// Library/POUs/Calculation/MC_CalculateInverseKinematic/Structures/CalculateInverseKinematicRecvData
{attribute 'pack_mode' := '1'} 
// ------------------------------------------------------------------------- 
//  SRCI Robot Library                                                
// ------------------------------------------------------------------------- 
//                                                                           
//  Object:      CalculateInverseKinematicRecvData                                       
//  Author:      Thorsten Brach                                                
//  Date:        2024-06-09
//
//  Description:                                              
//   
//                                                                           
//  Copyright: 
//    (C) 2024 Thorsten Brach. All rights reserved                                                                                                                                            
//             Licensed under the LGPL-3.0 license.
//                                                                           
//  Disclaimer:                                                                           
//    This project is provided without any guarantee and can be used for   
//    private and commercial purposes. Any use is at the user’s 
//    own risk and responsibility.
//
// -------------------------------------------------------------------------
TYPE CalculateInverseKinematicRecvData EXTENDS RspHeader :
STRUCT
  /// Calculated robot joint position
  JointPosition      : RobotJointPosition;  
END_STRUCT
END_TYPE

// Library/POUs/Calculation/MC_CalculateInverseKinematic/Structures/CalculateInverseKinematicSendData
{attribute 'pack_mode' := '1'}
// ------------------------------------------------------------------------- 
//  SRCI Robot Library                                                
// ------------------------------------------------------------------------- 
//                                                                           
//  Object:      CalculateInverseKinematicSendData                                       
//  Author:      Thorsten Brach                                                
//  Date:        2024-06-09
//
//  Description:                                              
//   
//                                                                           
//  Copyright: 
//    (C) 2024 Thorsten Brach. All rights reserved                                                                                                                                            
//             Licensed under the LGPL-3.0 license.
//                                                                           
//  Disclaimer:                                                                           
//    This project is provided without any guarantee and can be used for   
//    private and commercial purposes. Any use is at the user’s 
//    own risk and responsibility.
//
// -------------------------------------------------------------------------
TYPE CalculateInverseKinematicSendData EXTENDS CmdHeader:   
STRUCT
  /// cartesian position
  CartesianPosition  : RobotCartesianPosition;
  /// Index of target tool
  /// • 0: Flange (default)
  /// • 1..254: Tool frames
  ToolNo             : USINT;
  /// Index of target frame
  /// • 0: WCS (default)
  /// • 1..254: User frames
  FrameNo            : USINT;  
END_STRUCT
END_TYPE

// Library/POUs/Calculation/MC_CalculateTool/Structures/CalculateToolOutCmd
{attribute 'pack_mode' := '1'} 
// ------------------------------------------------------------------------- 
//  SRCI Robot Library                                                
// ------------------------------------------------------------------------- 
//                                                                           
//  Object:      CalculateToolOutCmd                                       
//  Author:      Thorsten Brach                                                
//  Date:        2024-06-09
//
//  Description:                                              
//   
//                                                                           
//  Copyright: 
//    (C) 2024 Thorsten Brach. All rights reserved                                                                                                                                                                                                               
//             Licensed under the LGPL-3.0 license.
//                                                                           
//  Disclaimer:                                                                           
//    This project is provided without any guarantee and can be used for   
//    private and commercial purposes. Any use is at the user’s 
//    own risk and responsibility.
//
// -------------------------------------------------------------------------
TYPE CalculateToolOutCmd :
STRUCT
  /// Tool data
  ToolData           : ToolData;
  /// Maximum error of deviation of the TCP position
  /// from the fix point in world coordinate system
  /// If not supported: • -1
  TCPMaxError       : REAL;
  /// Average error of TCP position from the fix point  in world coordinate system
  /// If not supported: • -1 
  TCPMeanError      : REAL;
END_STRUCT
END_TYPE

// Library/POUs/Calculation/MC_CalculateTool/Structures/CalculateToolParCmd
{attribute 'pack_mode' := '1'} 
// ------------------------------------------------------------------------- 
//  SRCI Robot Library                                                
// ------------------------------------------------------------------------- 
//                                                                           
//  Object:      CalculateToolParCmd                                       
//  Author:      Thorsten Brach                                                
//  Date:        2024-06-09
//
//  Description:                                              
//   
//                                                                           
//  Copyright: 
//    (C) 2024 Thorsten Brach. All rights reserved                                                                                                                                      
//             Licensed under the LGPL-3.0 license.
//                                                                           
//  Disclaimer:                                                                           
//    This project is provided without any guarantee and can be used for   
//    private and commercial purposes. Any use is at the user’s 
//    own risk and responsibility.
//
// -------------------------------------------------------------------------
TYPE CalculateToolParCmd :
STRUCT
  /// Define which method should be used to calculate the tool frame
  Mode               : ToolCalculationMode;
  /// Index of target tool
  /// • 0: Flange (default)
  /// • 1..254: Tool frames
  ToolNo             : USINT;
  /// Index of target frame
  /// • 0: WCS (default)
  /// • 1..254: User frames
  FrameNo            : USINT;  
  /// • True: Tool fixed
  /// • False: Tool on flange (default)
  ExternalTCP        : BOOL;
  /// Positions in cartesian coordinates for the tool frame calculation.
  PositionsArray     : ARRAY[0..5] OF RobotCartesianPosition;
END_STRUCT
END_TYPE

// Library/POUs/Calculation/MC_CalculateTool/Structures/CalculateToolRecvData
{attribute 'pack_mode' := '1'} 
// ------------------------------------------------------------------------- 
//  SRCI Robot Library                                                
// ------------------------------------------------------------------------- 
//                                                                           
//  Object:      CalculateToolRecvData                                       
//  Author:      Thorsten Brach                                                
//  Date:        2024-06-09
//
//  Description:                                              
//   
//                                                                           
//  Copyright: 
//    (C) 2024 Thorsten Brach. All rights reserved                                                                                                                                            
//             Licensed under the LGPL-3.0 license.
//                                                                           
//  Disclaimer:                                                                           
//    This project is provided without any guarantee and can be used for   
//    private and commercial purposes. Any use is at the user’s 
//    own risk and responsibility.
//
// -------------------------------------------------------------------------
TYPE CalculateToolRecvData EXTENDS RspHeader :
STRUCT
  /// Maximum error of deviation of the TCP position
  /// from the fix point in world coordinate system
  /// If not supported: • -1
  TCPMaxError       : REAL;
  /// Average error of TCP position from the fix point  in world coordinate system
  /// If not supported: • -1 
  TCPMeanError      : REAL;
  /// Tool data
  ToolData           : ToolData;
END_STRUCT
END_TYPE

// Library/POUs/Calculation/MC_CalculateTool/Structures/CalculateToolSendData
{attribute 'pack_mode' := '1'}
// ------------------------------------------------------------------------- 
//  SRCI Robot Library                                                
// ------------------------------------------------------------------------- 
//                                                                           
//  Object:      CalculateToolSendData                                       
//  Author:      Thorsten Brach                                                
//  Date:        2024-06-09
//
//  Description:                                              
//   
//                                                                           
//  Copyright: 
//    (C) 2024 Thorsten Brach. All rights reserved                                                                                                                                            
//             Licensed under the LGPL-3.0 license.
//                                                                           
//  Disclaimer:                                                                           
//    This project is provided without any guarantee and can be used for   
//    private and commercial purposes. Any use is at the user’s 
//    own risk and responsibility.
//
// -------------------------------------------------------------------------
TYPE CalculateToolSendData EXTENDS CmdHeader:   
STRUCT
  DataIndex    : USINT;
  ///
  DataComplete : BYTE;
  /// Index of target tool
  /// • 0: Flange (default)
  /// • 1..254: Tool frames
  ToolNo       : USINT;
  /// Index of target frame
  /// • 0: WCS (default)
  /// • 1..254: User frames
  FrameNo      : USINT;    
  /// Define which method should be used to calculate the tool frame
  Mode         : ToolCalculationMode;
  /// • True: Tool fixed
  /// • False: Tool on flange (default)
  ExternalTCP  : USINT;
  /// Positions in cartesian coordinates for the tool frame calculation.
  Position     : RobotCartesianPosition;
END_STRUCT
END_TYPE

// Library/POUs/Calculation/MC_LoadMeasurementAutomatic/Structures/LoadMeasurementAutomaticOutCmd
{attribute 'pack_mode' := '1'} 
// ------------------------------------------------------------------------- 
//  SRCI Robot Library                                                
// ------------------------------------------------------------------------- 
//                                                                           
//  Object:      LoadMeasurementAutomaticOutCmd                                       
//  Author:      Thorsten Brach                                                
//  Date:        2024-06-20
//
//  Description:                                              
//   
//                                                                           
//  Copyright: 
//    (C) 2024 Thorsten Brach. All rights reserved                                                                                                                                            
//             Licensed under the LGPL-3.0 license.
//                                                                           
//  Disclaimer:                                                                           
//    This project is provided without any guarantee and can be used for   
//    private and commercial purposes. Any use is at the user’s 
//    own risk and responsibility.
//
// -------------------------------------------------------------------------
TYPE LoadMeasurementAutomaticOutCmd :
STRUCT
  /// FB is returning a unique ID for the cal led measurement.
  MeasuringID       : UINT;
  /// Measured load data (see chapter 5.5.6.4)
  LoadData          : LoadData;  
  /// Load data available
  LoadDataAvailable : BOOL;
END_STRUCT
END_TYPE

// Library/POUs/Calculation/MC_LoadMeasurementAutomatic/Structures/LoadMeasurementAutomaticParCmd
{attribute 'pack_mode' := '1'} 
// ------------------------------------------------------------------------- 
//  SRCI Robot Library                                                
// ------------------------------------------------------------------------- 
//                                                                           
//  Object:      LoadMeasurementAutomaticParCmd                                       
//  Author:      Thorsten Brach                                                
//  Date:        2024-06-20
//
//  Description:                                              
//   
//                                                                           
//  Copyright: 
//    (C) 2024 Thorsten Brach. All rights reserved                                                                                                                                            
//             Licensed under the LGPL-3.0 license.
//                                                                           
//  Disclaimer:                                                                           
//    This project is provided without any guarantee and can be used for   
//    private and commercial purposes. Any use is at the user’s 
//    own risk and responsibility.
//
// -------------------------------------------------------------------------
TYPE LoadMeasurementAutomaticParCmd :
STRUCT
  /// Define which method should be used to measure the load data
  Mode               : LoadMeasurementMode;
  /// Define which mass is expected as a result of the load measurement
  Mass               : REAL;
  /// Define the area for the allowed motion of the Joint 3. 
  /// The order of the two limit values does not matter. 
  /// Only considered with "Mode" = 0, 2.
  Area_J3            : ARRAY[0..1] OF REAL;
  /// Define the area for the allowed motion of the Joint 4. 
  /// The order of the two limit values does not matter. 
  /// Only considered with "Mode" = 0, 2.
  Area_J4            : ARRAY[0..1] OF REAL;
  /// Define the area for the allowed motion of the Joint 5. 
  /// The order of the two limit values does not matter. 
  /// Only considered with "Mode" = 0, 2.
  Area_J5            : ARRAY[0..1] OF REAL;
  /// Define the area for the allowed motion of the Joint 6. 
  /// The order of the two limit values does not matter. 
  /// Only considered with "Mode" = 0, 2.
  Area_J6            : ARRAY[0..1] OF REAL;
  /// Define the first position for the load measurement.
  /// Only considered with "Mode" = 0, 1.
  Position_1         : RobotJointPosition;
  /// Define the second position for the load measurement.
  /// Only considered with "Mode" = 3.
  Position_2         : RobotJointPosition;
  /// Define the configuration angle for the load measurement.
  /// Only considered with "Mode" = 1.
  ConfigurationAngle : REAL;
END_STRUCT
END_TYPE

// Library/POUs/Calculation/MC_LoadMeasurementAutomatic/Structures/LoadMeasurementAutomaticRecvData
{attribute 'pack_mode' := '1'} 
// ------------------------------------------------------------------------- 
//  SRCI Robot Library                                                
// ------------------------------------------------------------------------- 
//                                                                           
//  Object:      LoadMeasurementAutomaticRecvData                                       
//  Author:      Thorsten Brach                                                
//  Date:        2024-06-20
//
//  Description:                                              
//   
//                                                                           
//  Copyright: 
//    (C) 2024 Thorsten Brach. All rights reserved                                                                                                                                            
//             Licensed under the LGPL-3.0 license.
//                                                                           
//  Disclaimer:                                                                           
//    This project is provided without any guarantee and can be used for   
//    private and commercial purposes. Any use is at the user’s 
//    own risk and responsibility.
//
// -------------------------------------------------------------------------
TYPE LoadMeasurementAutomaticRecvData EXTENDS RspHeader :
STRUCT
    /// FB is returning a unique ID for the cal led measurement.
  MeasuringID       : UINT;
  /// Measured load data (see chapter 5.5.6.4)
  LoadData          : LoadData;  
  /// Load data available
  LoadDataAvailable : BOOL;
END_STRUCT
END_TYPE

// Library/POUs/Calculation/MC_LoadMeasurementAutomatic/Structures/LoadMeasurementAutomaticSendData
{attribute 'pack_mode' := '1'}
// ------------------------------------------------------------------------- 
//  SRCI Robot Library                                                
// ------------------------------------------------------------------------- 
//                                                                           
//  Object:      LoadMeasurementAutomaticSendData                                       
//  Author:      Thorsten Brach                                                
//  Date:        2024-06-20
//
//  Description:                                              
//   
//                                                                           
//  Copyright: 
//    (C) 2024 Thorsten Brach. All rights reserved                                                                                                                                            
//             Licensed under the LGPL-3.0 license.
//                                                                           
//  Disclaimer:                                                                           
//    This project is provided without any guarantee and can be used for   
//    private and commercial purposes. Any use is at the user’s 
//    own risk and responsibility.
//
// -------------------------------------------------------------------------
TYPE LoadMeasurementAutomaticSendData EXTENDS CmdHeader:   
STRUCT
    /// Define which mass is expected as a result of the load measurement
  Mass               : REAL;
  /// Define which method should be used to measure the load data
  Mode               : LoadMeasurementMode;
  /// Reserved
  Reserved           : BYTE;
  /// Define the area for the allowed motion of the Joint 3. 
  /// The order of the two limit values does not matter. 
  /// Only considered with "Mode" = 0, 2.
  Area_J3            : ARRAY[0..1] OF REAL;
  /// Define the area for the allowed motion of the Joint 4. 
  /// The order of the two limit values does not matter. 
  /// Only considered with "Mode" = 0, 2.
  Area_J4            : ARRAY[0..1] OF REAL;
  /// Define the area for the allowed motion of the Joint 5. 
  /// The order of the two limit values does not matter. 
  /// Only considered with "Mode" = 0, 2.
  Area_J5            : ARRAY[0..1] OF REAL;
  /// Define the area for the allowed motion of the Joint 6. 
  /// The order of the two limit values does not matter. 
  /// Only considered with "Mode" = 0, 2.
  Area_J6            : ARRAY[0..1] OF REAL;
  /// Define the configuration angle for the load measurement.
  /// Only considered with "Mode" = 1.
  ConfigurationAngle : REAL;
  /// Define the first position for the load measurement.
  /// Only considered with "Mode" = 0, 1.
  Position_1         : RobotJointPosition;
  /// Define the second position for the load measurement.
  /// Only considered with "Mode" = 3.
  Position_2         : RobotJointPosition;
END_STRUCT
END_TYPE

// Library/POUs/Calculation/MC_LoadMeasurementSequential/Structures/LoadMeasurementSequentialOutCmd
{attribute 'pack_mode' := '1'} 
// ------------------------------------------------------------------------- 
//  SRCI Robot Library                                                
// ------------------------------------------------------------------------- 
//                                                                           
//  Object:      LoadMeasurementSequentialOutCmd                                       
//  Author:      Thorsten Brach                                                
//  Date:        2024-06-20
//
//  Description:                                              
//   
//                                                                           
//  Copyright: 
//    (C) 2024 Thorsten Brach. All rights reserved                                                                                                                                            
//             Licensed under the LGPL-3.0 license.
//                                                                           
//  Disclaimer:                                                                           
//    This project is provided without any guarantee and can be used for   
//    private and commercial purposes. Any use is at the user’s 
//    own risk and responsibility.
//
// -------------------------------------------------------------------------
TYPE LoadMeasurementSequentialOutCmd :
STRUCT
  /// FB is returning a unique ID for the cal led measurement.
  MeasuringID        : UINT;
  /// Measured load data (see chapter 5.5.6.4)
  LoadData           : LoadData;
  /// Load data available
  LoadDataAvailable : BOOL;
END_STRUCT
END_TYPE

// Library/POUs/Calculation/MC_LoadMeasurementSequential/Structures/LoadMeasurementSequentialParCmd
{attribute 'pack_mode' := '1'} 
// ------------------------------------------------------------------------- 
//  SRCI Robot Library                                                
// ------------------------------------------------------------------------- 
//                                                                           
//  Object:      LoadMeasurementSequentialParCmd                                       
//  Author:      Thorsten Brach                                                
//  Date:        2024-06-20
//
//  Description:                                              
//   
//                                                                           
//  Copyright: 
//    (C) 2024 Thorsten Brach. All rights reserved                                                                                                                                            
//             Licensed under the LGPL-3.0 license.
//                                                                           
//  Disclaimer:                                                                           
//    This project is provided without any guarantee and can be used for   
//    private and commercial purposes. Any use is at the user’s 
//    own risk and responsibility.
//
// -------------------------------------------------------------------------
TYPE LoadMeasurementSequentialParCmd :
STRUCT
  /// Define which step of the load estimation should be executed:
  Mode               : LoadMeasurementSteps;
  /// Define which mass is expected as a result of the load measurement
  Mass               : REAL;
END_STRUCT
END_TYPE

// Library/POUs/Calculation/MC_LoadMeasurementSequential/Structures/LoadMeasurementSequentialRecvData
{attribute 'pack_mode' := '1'} 
// ------------------------------------------------------------------------- 
//  SRCI Robot Library                                                
// ------------------------------------------------------------------------- 
//                                                                           
//  Object:      LoadMeasurementSequentialRecvData                                       
//  Author:      Thorsten Brach                                                
//  Date:        2024-06-20
//
//  Description:                                              
//   
//                                                                           
//  Copyright: 
//    (C) 2024 Thorsten Brach. All rights reserved                                                                                                                                            
//             Licensed under the LGPL-3.0 license.
//                                                                           
//  Disclaimer:                                                                           
//    This project is provided without any guarantee and can be used for   
//    private and commercial purposes. Any use is at the user’s 
//    own risk and responsibility.
//
// -------------------------------------------------------------------------
TYPE LoadMeasurementSequentialRecvData EXTENDS RspHeader :
STRUCT
  /// FB is returning a unique ID for the cal led measurement.
  MeasuringID       : UINT;
  /// Measured load data (see chapter 5.5.6.4)
  LoadData          : LoadData;  
  /// Load data available
  LoadDataAvailable : BOOL;
END_STRUCT
END_TYPE

// Library/POUs/Calculation/MC_LoadMeasurementSequential/Structures/LoadMeasurementSequentialSendData
{attribute 'pack_mode' := '1'}
// ------------------------------------------------------------------------- 
//  SRCI Robot Library                                                
// ------------------------------------------------------------------------- 
//                                                                           
//  Object:      LoadMeasurementSequentialSendData                                       
//  Author:      Thorsten Brach                                                
//  Date:        2024-06-20
//
//  Description:                                              
//   
//                                                                           
//  Copyright: 
//    (C) 2024 Thorsten Brach. All rights reserved                                                                                                                                            
//             Licensed under the LGPL-3.0 license.
//                                                                           
//  Disclaimer:                                                                           
//    This project is provided without any guarantee and can be used for   
//    private and commercial purposes. Any use is at the user’s 
//    own risk and responsibility.
//
// -------------------------------------------------------------------------
TYPE LoadMeasurementSequentialSendData EXTENDS CmdHeader:   
STRUCT
    /// Define which mass is expected as a result of the load measurement
  Mass               : REAL;
  /// Define which step of the load estimation should be executed:
  Mode               : LoadMeasurementSteps;
END_STRUCT
END_TYPE

// Library/POUs/ConveyorTracking/MC_ActivateConveyorTracking/Structures/ActivateConveyorTrackingOutCmd
{attribute 'pack_mode' := '1'} 
// ------------------------------------------------------------------------- 
//  SRCI Robot Library                                                
// ------------------------------------------------------------------------- 
//                                                                           
//  Object:      ActivateConveyorTrackingOutCmd                                       
//  Author:      Thorsten Brach                                                
//  Date:        2024-06-11
//
//  Description:                                              
//   
//                                                                           
//  Copyright: 
//    (C) 2024 Thorsten Brach. All rights reserved                                                                                                                                                                                                               
//             Licensed under the LGPL-3.0 license.
//                                                                           
//  Disclaimer:                                                                           
//    This project is provided without any guarantee and can be used for   
//    private and commercial purposes. Any use is at the user’s 
//    own risk and responsibility.
//
// -------------------------------------------------------------------------
TYPE ActivateConveyorTrackingOutCmd :
STRUCT
  /// Current status of "ConveyorTracking" according to Table 6-432
  TrackingStatus     : TrackingStatus;
  /// Relates to "ConnectionMode" 1 – "RC connected": Traveled distance of assigned conveyor since ConveyorTracking has been activated (offset)
  RCEncoderValue     : REAL;
END_STRUCT
END_TYPE

// Library/POUs/ConveyorTracking/MC_ActivateConveyorTracking/Structures/ActivateConveyorTrackingParCmd
{attribute 'pack_mode' := '1'} 
// ------------------------------------------------------------------------- 
//  SRCI Robot Library                                                
// ------------------------------------------------------------------------- 
//                                                                           
//  Object:      ActivateConveyorTrackingParCmd                                       
//  Author:      Thorsten Brach                                                
//  Date:        2024-06-11
//
//  Description:                                              
//   
//                                                                           
//  Copyright: 
//    (C) 2024 Thorsten Brach. All rights reserved                                                                                                                                      
//             Licensed under the LGPL-3.0 license.
//                                                                           
//  Disclaimer:                                                                           
//    This project is provided without any guarantee and can be used for   
//    private and commercial purposes. Any use is at the user’s 
//    own risk and responsibility.
//
// -------------------------------------------------------------------------
TYPE ActivateConveyorTrackingParCmd :
STRUCT
  /// Index of assigned conveyor
  ConveyorNo         : SINT;
  /// Specifies encoder connection setup (at least one option must be supported)
  ConnectionMode     : ConnectionMode;
  /// Relates to "ConnectionMode" 1 – "PLC connected": Value of the encoder connected to the conveyor belt
  PLCEncoderValue    : REAL;
END_STRUCT
END_TYPE

// Library/POUs/ConveyorTracking/MC_ActivateConveyorTracking/Structures/ActivateConveyorTrackingRecvData
{attribute 'pack_mode' := '1'} 
// ------------------------------------------------------------------------- 
//  SRCI Robot Library                                                
// ------------------------------------------------------------------------- 
//                                                                           
//  Object:      ActivateConveyorTrackingRecvData                                       
//  Author:      Thorsten Brach                                                
//  Date:        2024-06-11
//
//  Description:                                              
//   
//                                                                           
//  Copyright: 
//    (C) 2024 Thorsten Brach. All rights reserved                                                                                                                                            
//             Licensed under the LGPL-3.0 license.
//                                                                           
//  Disclaimer:                                                                           
//    This project is provided without any guarantee and can be used for   
//    private and commercial purposes. Any use is at the user’s 
//    own risk and responsibility.
//
// -------------------------------------------------------------------------
TYPE ActivateConveyorTrackingRecvData EXTENDS RspHeader :
STRUCT
  /// Maximum error of deviation of the TCP position
  /// from the fix point in world coordinate system
  /// If not supported: • -1
  TrackingStatus : TrackingStatus;
END_STRUCT
END_TYPE

// Library/POUs/ConveyorTracking/MC_ActivateConveyorTracking/Structures/ActivateConveyorTrackingSendData
{attribute 'pack_mode' := '1'}
// ------------------------------------------------------------------------- 
//  SRCI Robot Library                                                
// ------------------------------------------------------------------------- 
//                                                                           
//  Object:      ActivateConveyorTrackingSendData                                       
//  Author:      Thorsten Brach                                                
//  Date:        2024-06-11
//
//  Description:                                              
//   
//                                                                           
//  Copyright: 
//    (C) 2024 Thorsten Brach. All rights reserved                                                                                                                                            
//             Licensed under the LGPL-3.0 license.
//                                                                           
//  Disclaimer:                                                                           
//    This project is provided without any guarantee and can be used for   
//    private and commercial purposes. Any use is at the user’s 
//    own risk and responsibility.
//
// -------------------------------------------------------------------------
TYPE ActivateConveyorTrackingSendData EXTENDS CmdHeader:   
STRUCT
  /// Index of assigned conveyor
  ConveyorNo     : SINT;
  /// Specifies encoder connection setup (at least one option must be supported)
  ConnectionMode : SINT;
END_STRUCT
END_TYPE

// Library/POUs/ConveyorTracking/MC_ConfigureConveyor/Structures/ConfigureConveyorOutCmd
{attribute 'pack_mode' := '1'} 
// ------------------------------------------------------------------------- 
//  SRCI Robot Library                                                
// ------------------------------------------------------------------------- 
//                                                                           
//  Object:      ConfigureConveyorOutCmd                                       
//  Author:      Thorsten Brach                                                
//  Date:        2024-06-11
//
//  Description:                                              
//   
//                                                                           
//  Copyright: 
//    (C) 2024 Thorsten Brach. All rights reserved                                                                                                                                                                                                               
//             Licensed under the LGPL-3.0 license.
//                                                                           
//  Disclaimer:                                                                           
//    This project is provided without any guarantee and can be used for   
//    private and commercial purposes. Any use is at the user’s 
//    own risk and responsibility.
//
// -------------------------------------------------------------------------
TYPE ConfigureConveyorOutCmd :
STRUCT
END_STRUCT
END_TYPE

// Library/POUs/ConveyorTracking/MC_ConfigureConveyor/Structures/ConfigureConveyorParCmd
{attribute 'pack_mode' := '1'} 
// ------------------------------------------------------------------------- 
//  SRCI Robot Library                                                
// ------------------------------------------------------------------------- 
//                                                                           
//  Object:      ConfigureConveyorParCmd                                       
//  Author:      Thorsten Brach                                                
//  Date:        2024-06-11
//
//  Description:                                              
//   
//                                                                           
//  Copyright: 
//    (C) 2024 Thorsten Brach. All rights reserved                                                                                                                                      
//             Licensed under the LGPL-3.0 license.
//                                                                           
//  Disclaimer:                                                                           
//    This project is provided without any guarantee and can be used for   
//    private and commercial purposes. Any use is at the user’s 
//    own risk and responsibility.
//
// -------------------------------------------------------------------------
TYPE ConfigureConveyorParCmd :
STRUCT
  /// Index of assigned conveyor
  ConveyorNo         : USINT;  
  ///Define the origin coordinate system of the conveyor belt, with the X-Axis pointing in the direction of the movement of the conveyor belt.
  ConveyorOrigin     : FrameData;
  /// Define the type of the conveyor
  ConveyorType       : ConveyorType;
  /// Relates to "ConveyorType" "Circular Tracking": Define the radius of the circular conveyor
  Radius             : REAL;
  /// Distance [mm] from the origin of the conveyor belt to the beginning of the "SyncInZone"
  StartDistance      : REAL;
  /// Distance [mm] from the origin of the conveyor belt to the end of the "SyncOutZone"
  EndDistance        : REAL;
  /// Define the length of the "SyncInZone"
  SyncInLength       : REAL;
  /// Define the length of the "SyncOutZone"
  SyncOutLength      : REAL;
END_STRUCT
END_TYPE

// Library/POUs/ConveyorTracking/MC_ConfigureConveyor/Structures/ConfigureConveyorRecvData
{attribute 'pack_mode' := '1'} 
// ------------------------------------------------------------------------- 
//  SRCI Robot Library                                                
// ------------------------------------------------------------------------- 
//                                                                           
//  Object:      ConfigureConveyorRecvData                                       
//  Author:      Thorsten Brach                                                
//  Date:        2024-06-11
//
//  Description:                                              
//   
//                                                                           
//  Copyright: 
//    (C) 2024 Thorsten Brach. All rights reserved                                                                                                                                            
//             Licensed under the LGPL-3.0 license.
//                                                                           
//  Disclaimer:                                                                           
//    This project is provided without any guarantee and can be used for   
//    private and commercial purposes. Any use is at the user’s 
//    own risk and responsibility.
//
// -------------------------------------------------------------------------
TYPE ConfigureConveyorRecvData EXTENDS RspHeader :
STRUCT
END_STRUCT
END_TYPE

// Library/POUs/ConveyorTracking/MC_ConfigureConveyor/Structures/ConfigureConveyorSendData
{attribute 'pack_mode' := '1'}
// ------------------------------------------------------------------------- 
//  SRCI Robot Library                                                
// ------------------------------------------------------------------------- 
//                                                                           
//  Object:      ConfigureConveyorSendData                                       
//  Author:      Thorsten Brach                                                
//  Date:        2024-06-11
//
//  Description:                                              
//   
//                                                                           
//  Copyright: 
//    (C) 2024 Thorsten Brach. All rights reserved                                                                                                                                            
//             Licensed under the LGPL-3.0 license.
//                                                                           
//  Disclaimer:                                                                           
//    This project is provided without any guarantee and can be used for   
//    private and commercial purposes. Any use is at the user’s 
//    own risk and responsibility.
//
// -------------------------------------------------------------------------
TYPE ConfigureConveyorSendData EXTENDS CmdHeader:   
STRUCT
  ///Define the origin coordinate system of the conveyor belt, with the X-Axis pointing in the direction of the movement of the conveyor belt.
  ConveyorOrigin          : FrameData;
  /// ConveyorOrigin available
  ConveyorOriginAvailable : BOOL;
  /// Index of assigned conveyor
  ConveyorNo              : USINT;  
  /// Define the type of the conveyor
  ConveyorType            : ConveyorType;
  /// Relates to "ConveyorType" "Circular Tracking": Define the radius of the circular conveyor
  Radius                  : REAL;
  /// Distance [mm] from the origin of the conveyor belt to the beginning of the "SyncInZone"
  StartDistance           : REAL;
  /// Distance [mm] from the origin of the conveyor belt to the end of the "SyncOutZone"
  EndDistance             : REAL;
  /// Define the length of the "SyncInZone"
  SyncInLength            : REAL;
  /// Define the length of the "SyncOutZone"
  SyncOutLength           : REAL;
END_STRUCT
END_TYPE

// Library/POUs/ConveyorTracking/MC_RedefineTrackingPos/Structures/RedefineTrackingPosOutCmd
{attribute 'pack_mode' := '1'} 
// ------------------------------------------------------------------------- 
//  SRCI Robot Library                                                
// ------------------------------------------------------------------------- 
//                                                                           
//  Object:      RedefineTrackingPosOutCmd                                       
//  Author:      Thorsten Brach                                                
//  Date:        2024-06-11
//
//  Description:                                              
//   
//                                                                           
//  Copyright: 
//    (C) 2024 Thorsten Brach. All rights reserved                                                                                                                                                                                                               
//             Licensed under the LGPL-3.0 license.
//                                                                           
//  Disclaimer:                                                                           
//    This project is provided without any guarantee and can be used for   
//    private and commercial purposes. Any use is at the user’s 
//    own risk and responsibility.
//
// -------------------------------------------------------------------------
TYPE RedefineTrackingPosOutCmd :
STRUCT
  /// Unique system-generated ID of the "Action" when the function is triggered.
  /// • >0: The "Action" is started by the trigger funcrion with identical FollowID.
  /// • <0: The "Action" is stopped by the trigger function with identical FollowID.
  /// For more information see chapter 5.5.12.4 EmitterID, ListenerID, FollowID and OriginID
  OriginID               : INT;
  /// Relates to ListenerID >0
  /// Number of successful trigger-based command invocations - For more information refer TO chapter 5.5.12.4
  InvocationCounter      : USINT;  
END_STRUCT
END_TYPE

// Library/POUs/ConveyorTracking/MC_RedefineTrackingPos/Structures/RedefineTrackingPosParCmd
{attribute 'pack_mode' := '1'} 
// ------------------------------------------------------------------------- 
//  SRCI Robot Library                                                
// ------------------------------------------------------------------------- 
//                                                                           
//  Object:      RedefineTrackingPosParCmd                                       
//  Author:      Thorsten Brach                                                
//  Date:        2024-06-11
//
//  Description:                                              
//   
//                                                                           
//  Copyright: 
//    (C) 2024 Thorsten Brach. All rights reserved                                                                                                                                      
//             Licensed under the LGPL-3.0 license.
//                                                                           
//  Disclaimer:                                                                           
//    This project is provided without any guarantee and can be used for   
//    private and commercial purposes. Any use is at the user’s 
//    own risk and responsibility.
//
// -------------------------------------------------------------------------
TYPE RedefineTrackingPosParCmd :
STRUCT
  /// Relates to ListenerID >0:
  ProcessingMode         : ProcessingMode;
  /// Index of assigned conveyor
  ConveyorNo             : USINT;
  /// Relates to ListenerID = 0:
  /// Define initial work piece position relative to the conveyor belt origin:
  /// • Origin (X, Y, Z in mm)
  /// • Orientation (RX, RY, RZ in degree)
  /// For more information refer to chapter 5.5.14.
  InitObjectPosition     : ARRAY[0..5] OF REAL;
  /// Relates to ListenerID = 0:
  /// Travel distance of assigned UCS between work piece detection (InitObjectPosition) and execution of this command.
  TrackingOffset         : REAL;
  /// Relates to ListenerID >0
  /// Start index of real registers containing InitObjectPosition for trigger-based execution.
  StartIndexInitPosition : USINT;
  /// Define the index number of the UCS that is assigned to the conveyor by the function "ConveyorTracking".
  /// For more information refer to chapter 5.5.14.
  FrameNo                : USINT;
  /// Relates to ListenerID >0
  /// Index of real register containing TrackingOffset for trigger-based execution
  IndexTrackingOffset    : USINT;
  /// ID of associated trigger function:
  /// • 0: No Trigger (default): No trigger related behavior
  /// • >0: Trigger: o Start executing, when the trigger function with the identical EmitterID is triggered.
  /// Always positive.
  /// For more information, see chapter 5.5.12 Triggers
  ListenerID             :  SINT;
END_STRUCT
END_TYPE

// Library/POUs/ConveyorTracking/MC_RedefineTrackingPos/Structures/RedefineTrackingPosRecvData
{attribute 'pack_mode' := '1'} 
// ------------------------------------------------------------------------- 
//  SRCI Robot Library                                                
// ------------------------------------------------------------------------- 
//                                                                           
//  Object:      RedefineTrackingPosRecvData                                       
//  Author:      Thorsten Brach                                                
//  Date:        2024-06-11
//
//  Description:                                              
//   
//                                                                           
//  Copyright: 
//    (C) 2024 Thorsten Brach. All rights reserved                                                                                                                                            
//             Licensed under the LGPL-3.0 license.
//                                                                           
//  Disclaimer:                                                                           
//    This project is provided without any guarantee and can be used for   
//    private and commercial purposes. Any use is at the user’s 
//    own risk and responsibility.
//
// -------------------------------------------------------------------------
TYPE RedefineTrackingPosRecvData EXTENDS RspHeader :
STRUCT
  
  InvocationCounter : USINT;
  /// Reserve
  Reserved          : SINT;
  /// Unique system-generated ID of the "Action" when the function is triggered.
  /// • >0: The "Action" is started by the trigger funcrion with identical FollowID.
  /// • <0: The "Action" is stopped by the trigger function with identical FollowID.
  /// For more information see chapter 5.5.12.4 EmitterID, ListenerID, FollowID and OriginID
  OriginID          : INT;
END_STRUCT
END_TYPE

// Library/POUs/ConveyorTracking/MC_RedefineTrackingPos/Structures/RedefineTrackingPosSendData
{attribute 'pack_mode' := '1'}
// ------------------------------------------------------------------------- 
//  SRCI Robot Library                                                
// ------------------------------------------------------------------------- 
//                                                                           
//  Object:      RedefineTrackingPosSendData                                       
//  Author:      Thorsten Brach                                                
//  Date:        2024-06-11
//
//  Description:                                              
//   
//                                                                           
//  Copyright: 
//    (C) 2024 Thorsten Brach. All rights reserved                                                                                                                                            
//             Licensed under the LGPL-3.0 license.
//                                                                           
//  Disclaimer:                                                                           
//    This project is provided without any guarantee and can be used for   
//    private and commercial purposes. Any use is at the user’s 
//    own risk and responsibility.
//
// -------------------------------------------------------------------------
TYPE RedefineTrackingPosSendData EXTENDS CmdHeader:   
STRUCT
  /// EmitterID
  EmitterID              : ARRAY[0..3] OF SINT;
  /// ID of associated trigger function:
  /// • 0: No Trigger (default): No trigger related behavior
  /// • >0: Trigger: o Start executing, when the trigger function with the identical EmitterID is triggered.
  /// Always positive.
  /// For more information, see chapter 5.5.12 Triggers
  ListenerID             : SINT;
  /// Reserve
  Reserve                : BYTE;
  /// Index of assigned conveyor
  ConveyorNo             : USINT;
  /// Relates to ListenerID >0
  /// Start index of real registers containing InitObjectPosition for trigger-based execution.
  StartIndexInitPosition : USINT;
  /// Relates to ListenerID = 0:
  /// Travel distance of assigned UCS between work piece detection (InitObjectPosition) and execution of this command.
  TrackingOffset         : REAL;
  /// Define the index number of the UCS that is assigned to the conveyor by the function "ConveyorTracking".
  /// For more information refer to chapter 5.5.14.
  FrameNo                : USINT;
  /// Relates to ListenerID >0
  /// Index of real register containing TrackingOffset for trigger-based execution
  IndexTrackingOffset    : USINT;
END_STRUCT
END_TYPE

// Library/POUs/ConveyorTracking/MC_SyncToConveyor/Structures/SyncToConveyorOutCmd
{attribute 'pack_mode' := '1'} 
// ------------------------------------------------------------------------- 
//  SRCI Robot Library                                                
// ------------------------------------------------------------------------- 
//                                                                           
//  Object:      SyncToConveyorOutCmd                                       
//  Author:      Thorsten Brach                                                
//  Date:        2024-06-11
//
//  Description:                                              
//   
//                                                                           
//  Copyright: 
//    (C) 2024 Thorsten Brach. All rights reserved                                                                                                                                                                                                               
//             Licensed under the LGPL-3.0 license.
//                                                                           
//  Disclaimer:                                                                           
//    This project is provided without any guarantee and can be used for   
//    private and commercial purposes. Any use is at the user’s 
//    own risk and responsibility.
//
// -------------------------------------------------------------------------
TYPE SyncToConveyorOutCmd :
STRUCT
  /// Relates to ListenerID >0
  /// Number of successful trigger-based command invocations - For more information refer TO chapter 5.5.12.4
  InvocationCounter      : USINT;  
  /// Reserve
  Reserve                : BYTE;
  /// Unique system-generated ID of the "Action" when the function is triggered.
  /// • >0: The "Action" is started by the trigger funcrion with identical FollowID.
  /// • <0: The "Action" is stopped by the trigger function with identical FollowID.
  /// For more information see chapter 5.5.12.4 EmitterID, ListenerID, FollowID and OriginID
  OriginID               : INT;
  /// The TCP is in synchronization with the object on the conveyor belt.
  InSync                 : BOOL;
END_STRUCT
END_TYPE

// Library/POUs/ConveyorTracking/MC_SyncToConveyor/Structures/SyncToConveyorParCmd
{attribute 'pack_mode' := '1'} 
// ------------------------------------------------------------------------- 
//  SRCI Robot Library                                                
// ------------------------------------------------------------------------- 
//                                                                           
//  Object:      SyncToConveyorParCmd                                       
//  Author:      Thorsten Brach                                                
//  Date:        2024-06-11
//
//  Description:                                              
//   
//                                                                           
//  Copyright: 
//    (C) 2024 Thorsten Brach. All rights reserved                                                                                                                                      
//             Licensed under the LGPL-3.0 license.
//                                                                           
//  Disclaimer:                                                                           
//    This project is provided without any guarantee and can be used for   
//    private and commercial purposes. Any use is at the user’s 
//    own risk and responsibility.
//
// -------------------------------------------------------------------------
TYPE SyncToConveyorParCmd :
STRUCT
  /// Index of assigned conveyor
  ConveyorNo      : USINT;
  /// Define the index number of the UCS that will be assigned to the conveyor.
  /// For more information refer to chapter 5.5.14
  FrameNo         : USINT;
  /// Defines when synchronization starts.
  SyncInMode      : SyncInMode;
  /// Relates to "SyncInMode" "After distance" (1) and "After time" (2):
  /// Parameter for the synchronization
  /// • "After distance" (1)
  ///    •  Distance in mm
  /// • "After time" (2)
  ////   • Time in ms
  SyncInParameter : REAL;
  /// Define the maximum adjustment velocity for the robot to catch up to the conveyor belt.
  /// The velocity must be greater than the velocity of the conveyor belt.
  /// • 0 (default): no limit
  ///       o No conveyor tracking specific limit
  ///       o RC internal limit applies
  /// • >0: use limit
  ///       o Conveyor tracking specific limit applies
  MaxVelocity     : REAL;
  /// Define the maximum adjustment acceleration for the robot to catch up to the conveyor belt.
  /// • 0 (default): no limit
  ///     o No conveyor tracking specific limit
  ///     o RC internal limit applies
  /// • >0: use limit
  ///     o Conveyor tracking specific limit applies
  MaxAcceleration : REAL;
  /// ID of associated trigger function:
  ///  •  0: No Trigger (default):
  ///        o No trigger related behavior
  ///  • >0: Trigger:
  ///        o Start executing, when the trigger function with the identical EmitterID is triggered.
  /// Always positive.
  /// For more information, see chapter 5.5.12 Triggers
  ListenerID      : SINT;
END_STRUCT
END_TYPE

// Library/POUs/ConveyorTracking/MC_SyncToConveyor/Structures/SyncToConveyorRecvData
{attribute 'pack_mode' := '1'} 
// ------------------------------------------------------------------------- 
//  SRCI Robot Library                                                
// ------------------------------------------------------------------------- 
//                                                                           
//  Object:      SyncToConveyorRecvData                                       
//  Author:      Thorsten Brach                                                
//  Date:        2024-06-11
//
//  Description:                                              
//   
//                                                                           
//  Copyright: 
//    (C) 2024 Thorsten Brach. All rights reserved                                                                                                                                            
//             Licensed under the LGPL-3.0 license.
//                                                                           
//  Disclaimer:                                                                           
//    This project is provided without any guarantee and can be used for   
//    private and commercial purposes. Any use is at the user’s 
//    own risk and responsibility.
//
// -------------------------------------------------------------------------
TYPE SyncToConveyorRecvData EXTENDS RspHeader :
STRUCT
  InvocationCounter : USINT;
  /// Reserve
  Reserved          : SINT;
  /// Unique system-generated ID of the "Action" when the function is triggered.
  /// • >0: The "Action" is started by the trigger funcrion with identical FollowID.
  /// • <0: The "Action" is stopped by the trigger function with identical FollowID.
  /// For more information see chapter 5.5.12.4 EmitterID, ListenerID, FollowID and OriginID
  OriginID          : INT;
  /// The TCP is in synchronization with the object on the conveyor belt.
  InSync            : BOOL;
END_STRUCT
END_TYPE

// Library/POUs/ConveyorTracking/MC_SyncToConveyor/Structures/SyncToConveyorSendData
{attribute 'pack_mode' := '1'}
// ------------------------------------------------------------------------- 
//  SRCI Robot Library                                                
// ------------------------------------------------------------------------- 
//                                                                           
//  Object:      SyncToConveyorSendData                                       
//  Author:      Thorsten Brach                                                
//  Date:        2024-06-11
//
//  Description:                                              
//   
//                                                                           
//  Copyright: 
//    (C) 2024 Thorsten Brach. All rights reserved                                                                                                                                            
//             Licensed under the LGPL-3.0 license.
//                                                                           
//  Disclaimer:                                                                           
//    This project is provided without any guarantee and can be used for   
//    private and commercial purposes. Any use is at the user’s 
//    own risk and responsibility.
//
// -------------------------------------------------------------------------
TYPE SyncToConveyorSendData EXTENDS CmdHeader:   
STRUCT
  /// EmitterID
  EmitterID       : ARRAY[0..3] OF SINT;
  /// ID of associated trigger function:
  /// • 0: No Trigger (default): No trigger related behavior
  /// • >0: Trigger: o Start executing, when the trigger function with the identical EmitterID is triggered.
  /// Always positive.
  /// For more information, see chapter 5.5.12 Triggers
  ListenerID      : SINT;
  /// Reserve
  Reserve         : BYTE;
  /// Index of assigned conveyor
  ConveyorNo      : USINT;
  /// Define the index number of the UCS that will be assigned to the conveyor.
  /// For more information refer to chapter 5.5.14
  FrameNo         : USINT;
  /// Defines when synchronization starts
  SyncInMode      : SyncInMode;
  /// Relates to "SyncInMode" "After distance" (1) and "After time" (2): Parameter for the synchronization
  /// • "After distance" (1) -  Distance in mm
  /// • "After time" (2) -  Time in ms
  SyncInParameter : REAL;
  /// Define the maximum adjustment velocity for the robot to catch up to the conveyor belt.
  /// The velocity must be greater than the velocity of the conveyor belt.
  /// • 0 (default): no limit - No conveyor tracking specific limit
  ///                         - RC internal limit applies
  /// • >0: use limit         - Conveyor tracking specific limit applies
  MaxVelocity     : REAL;
  /// Define the maximum adjustment acceleration for the robot to catch up to the conveyor belt.
  /// • 0 (default): no limit - No conveyor tracking specific limit
  ///                         - RC internal limit applies
  /// • >0: use limit         - Conveyor tracking specific limit applies
  MaxAcceleration : REAL;
  /// ID of associated trigger function:
  /// • 0: No Trigger (default): No trigger related behavior
  /// • >0: Trigger:  Start executing, when the trigger function with the identical EmitterID is triggered.
  /// Always positive.
  /// For more information, see chapter 5.5.12 Triggers
END_STRUCT
END_TYPE

// Library/POUs/ForceControl/MC_ForceControl/Structures/ForceControlOutCmd
{attribute 'pack_mode' := '1'} 
// ------------------------------------------------------------------------- 
//  SRCI Robot Library                                                
// ------------------------------------------------------------------------- 
//                                                                           
//  Object:      ForceControlOutCmd                                       
//  Author:      Thorsten Brach                                                
//  Date:        2024-06-16
//
//  Description:                                              
//   
//                                                                           
//  Copyright: 
//    (C) 2024 Thorsten Brach. All rights reserved                                                                                                                                                                                                               
//             Licensed under the LGPL-3.0 license.
//                                                                           
//  Disclaimer:                                                                           
//    This project is provided without any guarantee and can be used for   
//    private and commercial purposes. Any use is at the user’s 
//    own risk and responsibility.
//
// -------------------------------------------------------------------------
TYPE ForceControlOutCmd :
STRUCT
  /// Current status of ForceControl and ForceLimit (chapter 6.5.25) according to Table 6-712
  ForceStatus        : ForceStatus;  
END_STRUCT
END_TYPE

// Library/POUs/ForceControl/MC_ForceControl/Structures/ForceControlParCmd
{attribute 'pack_mode' := '1'} 
// ------------------------------------------------------------------------- 
//  SRCI Robot Library                                                
// ------------------------------------------------------------------------- 
//                                                                           
//  Object:      ForceControlParCmd                                       
//  Author:      Thorsten Brach                                                
//  Date:        2024-06-16
//
//  Description:                                              
//   
//                                                                           
//  Copyright: 
//    (C) 2024 Thorsten Brach. All rights reserved                                                                                                                                      
//             Licensed under the LGPL-3.0 license.
//                                                                           
//  Disclaimer:                                                                           
//    This project is provided without any guarantee and can be used for   
//    private and commercial purposes. Any use is at the user’s 
//    own risk and responsibility.
//
// -------------------------------------------------------------------------
TYPE ForceControlParCmd :
STRUCT
  /// Defines type of reference of Force and Torque (at least one option must be supported)
  ReferenceType      : ReferenceType;
  /// Relates to ConnectionMode 1 and 2 (Sensor connected to PLC).
  /// Currently applied force and torque detected by sensor according to ReferenceType, ToolNo and FrameNo.
  /// • [0]: X-Axis
  /// • [1]: Y-Axis
  /// • [2]: Z- Axis
  /// • [3]: Rotation around X-Axis (RX)
  /// • [4]: Rotation around Y-Axis (RY)
  /// • [5]: Rotation around Z- Axis (RZ)
  SensorValue        : ARRAY[0..5] OF REAL;
  /// Relates to ReferenceType 0 (Tool) and 1 (Frame):
  /// Force and torque to be applied by robot arm according to ReferenceType, ToolNo and FrameNo:
  /// • [0]: X-Axis
  /// • [1]: Y-Axis
  /// • [2]: Z- Axis
  /// • [3]: Rotation around X-Axis (RX)
  /// • [4]: Rotation around Y-Axis (RY)
  /// • [5]: Rotation around Z- Axis (RZ)
  /// Set TargetValue <>-99999.9999 (default) to define setpoint
  TargetValue        : ARRAY[0..5] OF REAL;
  /// Index of tool
  /// •      0: Flange (default)
  /// • 1..254: Tool frames
  ToolNo             : USINT;
  /// Define the index number of the UCS that will be assigned to the conveyor.
  /// For more information refer to chapter 5.5.14
  FrameNo            : USINT;
  /// Specifies encoder connection setup according to Table 6-713 (at least one option must be supported) 
  ConnectionMode     : SensorConnectionMode;
  /// Position of sensor relative to flange (FixedSensor FALSE) or relative to WCS (FixedSensor TRUE)
  /// • [0]: X-Axis
  /// • [1]: Y-Axis
  /// • [2]: Z- Axis
  /// • [3]: Rotation around X-Axis (RX)
  /// • [4]: Rotation around Y-Axis (RY)
  /// • [5]: Rotation around Z- Axis (RZ)
  SensorFrame        : ARRAY[0..5] OF REAL;
  /// Index of payload data containing mass, center of gravity, orientation and inertia relative to SensorFrame.
  /// Required to calibrate system for setting up gravity compensation and sensor offset.
  CalibrationData    : USINT;
  /// Tolerance of TargetValue within which currently applied force/torque will return ForceStatus "Specified force/torque reached" TRUE.
  TargetWindow       : REAL;
  /// Define axes whose position may be adjusted by the robot to apply specified force according to Table 6-711.
  CompliantAxes      : BYTE;
  /// Maximum allowed TCP velocity for compliant axes in % of nominal velocity.
  /// •   0% (default): no limit - RC internal limit applies
  /// •  >0% use limit -  Specified limit applies
  /// • 100% use maximal reference velocity
  /// For more information on nominal dynamics see chapter 5.5.7 Robot dynamics 
  MaxVelocity        : UINT;
  /// Maximum allowed cartesian deviation according to ReferenceType, ToolNo and FrameNo.
  /// Set 0 (default) to not specify a limit in this axis direction.
  /// • [0]: Deviation in X-Direction in mm
  /// • [1]: Deviation in Y- direction in mm
  /// • [2]: Deviation in Z- direction in mm
  /// • [3]: Deviation in RX- direction in °
  /// • [4]: Deviation in RY- direction in °
  /// • [5]: Deviation in RZ- direction in °
  MaxDeviation       : ARRAY [0..5] OF REAL;
  /// Defines reaction in case ForceControl reports error during its execution
  /// Processing of active move command is continued without active ForceControl
  ErrorReaction      : ErrorReaction;
  /// Relates to ErrorReaction 0 (Abort and move). Defines type of reference coordinate system of ErrorVector
  ErrorReferenceType : ReferenceType;
  /// Relates to ErrorReaction 0 (Abort and move). Vector defining robot’s movement in case of
  /// incoming error according to ErrorReferenceType, ErrorToolNo and ErrorFrameNo.
  /// • [0]: X-Axis
  /// • [1]: Y-Axis
  /// • [2]: Z- Axis
  /// • [3]: Rotation around X-Axis (RX)
  /// • [4]: Rotation around Y-Axis (RY)
  /// • [5]: Rotation around Z-Axis (RZ)
  ErrorVector        : ARRAY [0..5] OF REAL;
  /// Relates to ErrorReaction 0 (Abort and move). Index of tool.
  /// • 0 (default): Flange
  /// • 1..254: Tool frames
  ErrorToolNo        : USINT;
  /// Relates to ErrorReferenceType 1 (Frame)
  /// •      0: WCS (default)
  /// • 1..254: User frames
  ErrorFrameNo       : USINT;
  /// Defines sensor positioning:
  /// • FALSE (default): Sensor mounted on flange
  /// • TRUE: Sensor fixed
  FixedSensor        : BOOL;
END_STRUCT
END_TYPE

// Library/POUs/ForceControl/MC_ForceControl/Structures/ForceControlRecvData
{attribute 'pack_mode' := '1'} 
// ------------------------------------------------------------------------- 
//  SRCI Robot Library                                                
// ------------------------------------------------------------------------- 
//                                                                           
//  Object:      ForceControlRecvData                                       
//  Author:      Thorsten Brach                                                
//  Date:        2024-06-11
//
//  Description:                                              
//   
//                                                                           
//  Copyright: 
//    (C) 2024 Thorsten Brach. All rights reserved                                                                                                                                            
//             Licensed under the LGPL-3.0 license.
//                                                                           
//  Disclaimer:                                                                           
//    This project is provided without any guarantee and can be used for   
//    private and commercial purposes. Any use is at the user’s 
//    own risk and responsibility.
//
// -------------------------------------------------------------------------
TYPE ForceControlRecvData EXTENDS RspHeader :
STRUCT
  /// Current status of ForceControl and ForceLimit (chapter 6.5.25) according to Table 6-712
  ForceStatus : BYTE;
END_STRUCT
END_TYPE

// Library/POUs/ForceControl/MC_ForceControl/Structures/ForceControlSendData
{attribute 'pack_mode' := '1'}
// ------------------------------------------------------------------------- 
//  SRCI Robot Library                                                
// ------------------------------------------------------------------------- 
//                                                                           
//  Object:      ForceControlSendData                                       
//  Author:      Thorsten Brach                                                
//  Date:        2024-06-11
//
//  Description:                                              
//   
//                                                                           
//  Copyright: 
//    (C) 2024 Thorsten Brach. All rights reserved                                                                                                                                            
//             Licensed under the LGPL-3.0 license.
//                                                                           
//  Disclaimer:                                                                           
//    This project is provided without any guarantee and can be used for   
//    private and commercial purposes. Any use is at the user’s 
//    own risk and responsibility.
//
// -------------------------------------------------------------------------
TYPE ForceControlSendData EXTENDS CmdHeader:   
STRUCT
  /// Index of tool
  /// •      0: Flange (default)
  /// • 1..254: Tool frames
  ToolNo             : USINT;
  /// Define the index number of the UCS that will be assigned to the conveyor.
  /// For more information refer to chapter 5.5.14
  FrameNo            : USINT;
  /// Specifies encoder connection setup according to Table 6-713 (at least one option must be supported) 
  ConnectionMode     : SensorConnectionMode;
  /// Defines sensor positioning:
  /// • FALSE (default): Sensor mounted on flange
  /// • TRUE: Sensor fixed
  FixedSensor        : BYTE;
  /// Position of sensor relative to flange (FixedSensor FALSE) or relative to WCS (FixedSensor TRUE)
  /// • [0]: X-Axis
  /// • [1]: Y-Axis
  /// • [2]: Z- Axis
  /// • [3]: Rotation around X-Axis (RX)
  /// • [4]: Rotation around Y-Axis (RY)
  /// • [5]: Rotation around Z- Axis (RZ)
  SensorFrame        : ARRAY[0..5] OF REAL;
  /// Index of payload data containing mass, center of gravity, orientation and inertia relative to SensorFrame.
  /// Required to calibrate system for setting up gravity compensation and sensor offset.
  CalibrationData    : USINT;
  /// Defines type of reference of Force and Torque (at least one option must be supported)
  ReferenceType      : ReferenceType;
  /// Relates to ConnectionMode 1 and 2 (Sensor connected to PLC).
  /// Currently applied force and torque detected by sensor according to ReferenceType, ToolNo and FrameNo.
  /// • [0]: X-Axis
  /// • [1]: Y-Axis
  /// • [2]: Z- Axis
  /// • [3]: Rotation around X-Axis (RX)
  /// • [4]: Rotation around Y-Axis (RY)
  /// • [5]: Rotation around Z- Axis (RZ)
  SensorValue        : ARRAY[0..5] OF REAL;
  /// Relates to ReferenceType 0 (Tool) and 1 (Frame):
  /// Force and torque to be applied by robot arm according to ReferenceType, ToolNo and FrameNo:
  /// • [0]: X-Axis
  /// • [1]: Y-Axis
  /// • [2]: Z- Axis
  /// • [3]: Rotation around X-Axis (RX)
  /// • [4]: Rotation around Y-Axis (RY)
  /// • [5]: Rotation around Z- Axis (RZ)
  /// Set TargetValue <>-99999.9999 (default) to define setpoint
  TargetValue        : ARRAY[0..5] OF REAL;
  /// Maximum allowed TCP velocity for compliant axes in % of nominal velocity.
  /// •   0% (default): no limit - RC internal limit applies
  /// •  >0% use limit -  Specified limit applies
  /// • 100% use maximal reference velocity
  /// For more information on nominal dynamics see chapter 5.5.7 Robot dynamics 
  MaxVelocity        : UINT;
  /// Maximum allowed cartesian deviation according to ReferenceType, ToolNo and FrameNo.
  /// Set 0 (default) to not specify a limit in this axis direction.
  /// • [0]: Deviation in X-Direction in mm
  /// • [1]: Deviation in Y- direction in mm
  /// • [2]: Deviation in Z- direction in mm
  /// • [3]: Deviation in RX- direction in °
  /// • [4]: Deviation in RY- direction in °
  /// • [5]: Deviation in RZ- direction in °
  MaxDeviation       : ARRAY [0..5] OF REAL;
  /// Defines reaction in case ForceControl reports error during its execution
  /// Processing of active move command is continued without active ForceControl
  ErrorReaction      : ErrorReaction;
  /// Relates to ErrorReaction 0 (Abort and move). Defines type of reference coordinate system of ErrorVector
  ErrorReferenceType : ReferenceType;
  /// Relates to ErrorReaction 0 (Abort and move). Vector defining robot’s movement in case of
  /// incoming error according to ErrorReferenceType, ErrorToolNo and ErrorFrameNo.
  /// • [0]: X-Axis
  /// • [1]: Y-Axis
  /// • [2]: Z- Axis
  /// • [3]: Rotation around X-Axis (RX)
  /// • [4]: Rotation around Y-Axis (RY)
  /// • [5]: Rotation around Z-Axis (RZ)
  ErrorVector        : ARRAY [0..5] OF REAL;
  /// Relates to ErrorReaction 0 (Abort and move). Index of tool.
  /// • 0 (default): Flange
  /// • 1..254: Tool frames
  ErrorToolNo        : USINT;
  /// Relates to ErrorReferenceType 1 (Frame)
  /// •      0: WCS (default)
  /// • 1..254: User frames
  ErrorFrameNo       : USINT;
  /// Define axes whose position may be adjusted by the robot to apply specified force according to Table 6-711.
  CompliantAxes      : BYTE;
END_STRUCT
END_TYPE

// Library/POUs/ForceControl/MC_ForceLimit/Structures/ForceLimitOutCmd
{attribute 'pack_mode' := '1'} 
// ------------------------------------------------------------------------- 
//  SRCI Robot Library                                                
// ------------------------------------------------------------------------- 
//                                                                           
//  Object:      ForceLimitOutCmd                                       
//  Author:      Thorsten Brach                                                
//  Date:        2024-06-16
//
//  Description:                                              
//   
//                                                                           
//  Copyright: 
//    (C) 2024 Thorsten Brach. All rights reserved                                                                                                                                                                                                               
//             Licensed under the LGPL-3.0 license.
//                                                                           
//  Disclaimer:                                                                           
//    This project is provided without any guarantee and can be used for   
//    private and commercial purposes. Any use is at the user’s 
//    own risk and responsibility.
//
// -------------------------------------------------------------------------
TYPE ForceLimitOutCmd :
STRUCT
  /// Current status of ForceControl and ForceLimit (chapter 6.5.25) according to Table 6-712
  ForceStatus        : ForceStatus;
  /// Relates to EmitterID <> 0: Unique system-generated ID of the trigger function when the function is called by user.
  /// For more information see chapter 5.5.12.4.
  FollowID           : DINT;  
END_STRUCT
END_TYPE

// Library/POUs/ForceControl/MC_ForceLimit/Structures/ForceLimitParCmd
{attribute 'pack_mode' := '1'} 
// ------------------------------------------------------------------------- 
//  SRCI Robot Library                                                
// ------------------------------------------------------------------------- 
//                                                                           
//  Object:      ForceLimitParCmd                                       
//  Author:      Thorsten Brach                                                
//  Date:        2024-06-16
//
//  Description:                                              
//   
//                                                                           
//  Copyright: 
//    (C) 2024 Thorsten Brach. All rights reserved                                                                                                                                      
//             Licensed under the LGPL-3.0 license.
//                                                                           
//  Disclaimer:                                                                           
//    This project is provided without any guarantee and can be used for   
//    private and commercial purposes. Any use is at the user’s 
//    own risk and responsibility.
//
// -------------------------------------------------------------------------
TYPE ForceLimitParCmd :
STRUCT
  /// Defines type of reference of Force and Torque (at least one option must be supported)
  ReferenceType      : ReferenceType;
  /// Relates to ConnectionMode 1 and 2 (Sensor connected to PLC).
  /// Currently applied force and torque detected by sensor according to ReferenceType, ToolNo and FrameNo.
  /// • [0]: X-Axis
  /// • [1]: Y-Axis
  /// • [2]: Z- Axis
  /// • [3]: Rotation around X-Axis (RX)
  /// • [4]: Rotation around Y-Axis (RY)
  /// • [5]: Rotation around Z- Axis (RZ)
  SensorValue        : ARRAY[0..5] OF REAL;
  /// Index of tool
  /// •      0: Flange (default)
  /// • 1..254: Tool frames
  ToolNo             : USINT;
  /// Define the index number of the UCS that will be assigned to the conveyor.
  /// For more information refer to chapter 5.5.14
  FrameNo            : USINT;
  /// Maximal allowed force and torque detected by the sensor according to ReferenceType and ToolNo/FrameNo before robot reacts according to ReactionMode.
  /// Set value <>0 (default) to monitor coordinate axes
  /// • [0]: X-Axis
  /// • [1]: Y-Axis
  /// • [2]: Z- Axis
  /// • [3]: Rotation around X-Axis (RX)
  /// • [4]: Rotation around Y-Axis (RY)
  /// • [5]: Rotation around Z- Axis (RZ)
  ForceLimit        : ARRAY[0..5] OF REAL;
  /// Specifies encoder connection setup according to Table 6-713 (at least one option must be supported) 
  ConnectionMode    : SensorConnectionMode;
  /// Position of sensor relative to flange (FixedSensor FALSE) or relative to WCS (FixedSensor TRUE)
  /// • [0]: X-Axis
  /// • [1]: Y-Axis
  /// • [2]: Z- Axis
  /// • [3]: Rotation around X-Axis (RX)
  /// • [4]: Rotation around Y-Axis (RY)
  /// • [5]: Rotation around Z- Axis (RZ)
  SensorFrame        : ARRAY[0..5] OF REAL;
  /// Index of payload data containing mass, center of gravity, orientation and inertia relative to SensorFrame.
  /// Required to calibrate system for setting up gravity compensation and sensor offset.
  CalibrationData    : USINT;
  /// Defines sensor positioning:
  /// • FALSE (default): Sensor mounted on flange
  /// • TRUE: Sensor fixed
  FixedSensor        : BOOL;
  /// ID of Action that will be executed when this command is active
  /// • >0: Start Action        - Start executing the Action function with the identical ListenerID.
  /// • <0: Stop Action         - Stop executing the Action function with the identical ListenerID.
  /// •  0: Undefined (default) - If no EmitterID is defined, the function returns an error message
  /// For more information see chapter 5.5.12.4
  EmitterID          : SINT;  
END_STRUCT
END_TYPE

// Library/POUs/ForceControl/MC_ForceLimit/Structures/ForceLimitRecvData
{attribute 'pack_mode' := '1'} 
// ------------------------------------------------------------------------- 
//  SRCI Robot Library                                                
// ------------------------------------------------------------------------- 
//                                                                           
//  Object:      ForceLimitRecvData                                       
//  Author:      Thorsten Brach                                                
//  Date:        2024-06-11
//
//  Description:                                              
//   
//                                                                           
//  Copyright: 
//    (C) 2024 Thorsten Brach. All rights reserved                                                                                                                                            
//             Licensed under the LGPL-3.0 license.
//                                                                           
//  Disclaimer:                                                                           
//    This project is provided without any guarantee and can be used for   
//    private and commercial purposes. Any use is at the user’s 
//    own risk and responsibility.
//
// -------------------------------------------------------------------------
TYPE ForceLimitRecvData EXTENDS RspHeader :
STRUCT
  InvocationCounter : USINT;
  /// Reserve
  Reserved          : SINT;
  /// Unique system-generated ID of the "Action" when the function is triggered.
  /// • >0: The "Action" is started by the trigger funcrion with identical FollowID.
  /// • <0: The "Action" is stopped by the trigger function with identical FollowID.
  /// For more information see chapter 5.5.12.4 EmitterID, ListenerID, FollowID and OriginID
  OriginID          : INT;
  /// Current status of ForceControl and ForceLimit (chapter 6.5.25) according to Table 6-712
  ForceStatus       : BYTE;
END_STRUCT
END_TYPE

// Library/POUs/ForceControl/MC_ForceLimit/Structures/ForceLimitSendData
{attribute 'pack_mode' := '1'}
// ------------------------------------------------------------------------- 
//  SRCI Robot Library                                                
// ------------------------------------------------------------------------- 
//                                                                           
//  Object:      ForceLimitSendData                                       
//  Author:      Thorsten Brach                                                
//  Date:        2024-06-11
//
//  Description:                                              
//   
//                                                                           
//  Copyright: 
//    (C) 2024 Thorsten Brach. All rights reserved                                                                                                                                            
//             Licensed under the LGPL-3.0 license.
//                                                                           
//  Disclaimer:                                                                           
//    This project is provided without any guarantee and can be used for   
//    private and commercial purposes. Any use is at the user’s 
//    own risk and responsibility.
//
// -------------------------------------------------------------------------
TYPE ForceLimitSendData EXTENDS CmdHeader:   
STRUCT
  /// ID of Action that will be executed when this command is active
  /// • >0: Start Action        - Start executing the Action function with the identical ListenerID.
  /// • <0: Stop Action         - Stop executing the Action function with the identical ListenerID.
  /// •  0: Undefined (default) - If no EmitterID is defined, the function returns an error message
  /// For more information see chapter 5.5.12.4
  EmitterID          : ARRAY [0..3] OF SINT;
  /// ListenerID
  ListenerID         : SINT; 
  /// Reserve
  Reserve            : BYTE; 
  /// Index of tool
  /// •      0: Flange (default)
  /// • 1..254: Tool frames
  ToolNo             : USINT;
  /// Define the index number of the UCS that will be assigned to the conveyor.
  /// For more information refer to chapter 5.5.14
  FrameNo            : USINT;
  /// Specifies encoder connection setup according to Table 6-713 (at least one option must be supported) 
  ConnectionMode     : SensorConnectionMode;
  /// Defines sensor positioning:
  /// • FALSE (default): Sensor mounted on flange
  /// • TRUE: Sensor fixed
  FixedSensor        : BYTE;
  /// Position of sensor relative to flange (FixedSensor FALSE) or relative to WCS (FixedSensor TRUE)
  /// • [0]: X-Axis
  /// • [1]: Y-Axis
  /// • [2]: Z- Axis
  /// • [3]: Rotation around X-Axis (RX)
  /// • [4]: Rotation around Y-Axis (RY)
  /// • [5]: Rotation around Z- Axis (RZ)
  SensorFrame        : ARRAY[0..5] OF REAL;

  /// Index of payload data containing mass, center of gravity, orientation and inertia relative to SensorFrame.
  /// Required to calibrate system for setting up gravity compensation and sensor offset.
  CalibrationData    : USINT;
  /// Defines type of reference of Force and Torque (at least one option must be supported)
  ReferenceType      : ReferenceType;

  /// Relates to ConnectionMode 1 and 2 (Sensor connected to PLC).
  /// Currently applied force and torque detected by sensor according to ReferenceType, ToolNo and FrameNo.
  /// • [0]: X-Axis
  /// • [1]: Y-Axis
  /// • [2]: Z- Axis
  /// • [3]: Rotation around X-Axis (RX)
  /// • [4]: Rotation around Y-Axis (RY)
  /// • [5]: Rotation around Z- Axis (RZ)
  SensorValue        : ARRAY[0..5] OF REAL;
  /// Maximal allowed force and torque detected by the sensor according to ReferenceType and ToolNo/FrameNo before robot reacts according to ReactionMode.
  /// Set value <>0 (default) to monitor coordinate axes
  /// • [0]: X-Axis
  /// • [1]: Y-Axis
  /// • [2]: Z- Axis
  /// • [3]: Rotation around X-Axis (RX)
  /// • [4]: Rotation around Y-Axis (RY)
  /// • [5]: Rotation around Z- Axis (RZ)
  ForceLimit        : ARRAY[0..5] OF REAL;  
END_STRUCT
END_TYPE

// Library/POUs/ForceControl/MC_ReadActualForce/Structures/ReadActualForceOutCmd
{attribute 'pack_mode' := '1'} 
// ------------------------------------------------------------------------- 
//  SRCI Robot Library                                                
// ------------------------------------------------------------------------- 
//                                                                           
//  Object:      ReadActualForceOutCmd                                       
//  Author:      Thorsten Brach                                                
//  Date:        2024-06-16
//
//  Description:                                              
//   
//                                                                           
//  Copyright: 
//    (C) 2024 Thorsten Brach. All rights reserved                                                                                                                                                                                                               
//             Licensed under the LGPL-3.0 license.
//                                                                           
//  Disclaimer:                                                                           
//    This project is provided without any guarantee and can be used for   
//    private and commercial purposes. Any use is at the user’s 
//    own risk and responsibility.
//
// -------------------------------------------------------------------------
TYPE ReadActualForceOutCmd :
STRUCT
  /// Currently detected force and torque according to ReferenceType, ToolNo and FrameNo.
  /// • [0]: X-Axis
  /// • [1]: Y-Axis
  /// • [2]: Z- Axis
  /// • [3]: Rotation around X-Axis (RX)
  /// • [4]: Rotation around Y-Axis (RY)
  /// • [5]: Rotation around Z- Axis (RZ)
  ActualForce        : ARRAY[0..5] OF REAL;
  /// Unique system-generated ID of the "Action" when the function is triggered.
  /// • >0: The "Action" is started by the trigger function with identical FollowID.
  /// • <0: The "Action" is stopped by the trigger function with identical FollowID.
  /// For more information see chapter 5.5.12.4 EmitterID, ListenerID, FollowID and OriginID
  OriginID           : INT;
  /// Relates to ListenerID >0
  /// Number of successful trigger -based command invocations
  /// For more information refer to chapter 5.5.12.4.
  InvocationCounter  : USINT;  
END_STRUCT
END_TYPE

// Library/POUs/ForceControl/MC_ReadActualForce/Structures/ReadActualForceParCmd
{attribute 'pack_mode' := '1'} 
// ------------------------------------------------------------------------- 
//  SRCI Robot Library                                                
// ------------------------------------------------------------------------- 
//                                                                           
//  Object:      ReadActualForceParCmd                                       
//  Author:      Thorsten Brach                                                
//  Date:        2024-06-16
//
//  Description:                                              
//   
//                                                                           
//  Copyright: 
//    (C) 2024 Thorsten Brach. All rights reserved                                                                                                                                      
//             Licensed under the LGPL-3.0 license.
//                                                                           
//  Disclaimer:                                                                           
//    This project is provided without any guarantee and can be used for   
//    private and commercial purposes. Any use is at the user’s 
//    own risk and responsibility.
//
// -------------------------------------------------------------------------
TYPE ReadActualForceParCmd :
STRUCT
  /// Processing Mode
  ProcessingMode      : ProcessingMode;
  /// Defines type of reference of Force and Torque (at least one option must be supported )
  ReferenceType       : ReferenceType;
  /// Index of tool
  /// •      0: Flange (default)
  /// • 1..254: Tool frames
  ToolNo             : USINT;
  /// Define the index number of the UCS that will be assigned to the conveyor.
  /// For more information refer to chapter 5.5.14
  FrameNo            : USINT;
  /// Index of payload data containing mass, center of gravity, orientation and inertia relative to SensorFrame.
  /// Required to calibrate system for setting up gravity compensation and sensor offset.
  CalibrationData    : USINT;
  /// ID of associated trigger function:
  /// • 0: Immediately (default) - Start executing this function immediately.
  /// • >0: Trigger -  Start executing, when the trigger function with the identical EmitterID is triggered.
  /// Always positive.
  /// For more information, see chapter 5.5.12 Triggers
  ListenerID         : SINT; 
END_STRUCT
END_TYPE

// Library/POUs/ForceControl/MC_ReadActualForce/Structures/ReadActualForceRecvData
{attribute 'pack_mode' := '1'} 
// ------------------------------------------------------------------------- 
//  SRCI Robot Library                                                
// ------------------------------------------------------------------------- 
//                                                                           
//  Object:      ReadActualForceRecvData                                       
//  Author:      Thorsten Brach                                                
//  Date:        2024-06-11
//
//  Description:                                              
//   
//                                                                           
//  Copyright: 
//    (C) 2024 Thorsten Brach. All rights reserved                                                                                                                                            
//             Licensed under the LGPL-3.0 license.
//                                                                           
//  Disclaimer:                                                                           
//    This project is provided without any guarantee and can be used for   
//    private and commercial purposes. Any use is at the user’s 
//    own risk and responsibility.
//
// -------------------------------------------------------------------------
TYPE ReadActualForceRecvData EXTENDS RspHeader :
STRUCT
  InvocationCounter : USINT;
  /// Reserve
  Reserved          : SINT;
  /// Unique system-generated ID of the "Action" when the function is triggered.
  /// • >0: The "Action" is started by the trigger funcrion with identical FollowID.
  /// • <0: The "Action" is stopped by the trigger function with identical FollowID.
  /// For more information see chapter 5.5.12.4 EmitterID, ListenerID, FollowID and OriginID
  OriginID          : INT;
  /// Currently detected force and torque according to ReferenceType, ToolNo and FrameNo.
  /// • [0]: X-Axis
  /// • [1]: Y-Axis
  /// • [2]: Z- Axis
  /// • [3]: Rotation around X-Axis (RX)
  /// • [4]: Rotation around Y-Axis (RY)
  /// • [5]: Rotation around Z- Axis (RZ)
  ActualForce       : ARRAY[0..5] OF REAL;
END_STRUCT
END_TYPE

